// Service for ingesting data. This function block should be called on 
// every cycle to continually stream any data stored in the internal buffer.
FUNCTION_BLOCK FB_IngestService
VAR_INPUT
	hSiftClient : REFERENCE TO T_SiftClient;
	sRunId : STRING(255);
	aFlowConfigs : POINTER TO ST_FlowConfig;
END_VAR

VAR_OUTPUT
	bError : BOOL;
	nErrId : UDINT;
	nMsgsSent : UDINT; // Number of total messages sent to sift_proxy.
	nBufSize : UDINT; // The number of messages in the buffer.
	fBufferUtilization : LREAL; // The percent utilization of the internal buffer.
END_VAR

VAR
	eState : (IDLE, SEND_MESSAGE, SEND_MESSAGE_WAIT, SUCCESS, FAILURE):= IDLE;
	fbSendRingBuffer : FB_MemRingBuffer;
	aSendRingBuffer : ARRAY[0..SiftClientParameters.MAX_PACKET_SIZE - 1] OF BYTE;
	aTmpBuffer : ARRAY[0..SiftClientParameters.MAX_PACKET_SIZE - 1] OF BYTE;
	curOffset : UDINT;
	i : UDINT;
	nCount : UDINT;
END_VAR

nBufSize := fbSendRingBuffer.nCount;
fBufferUtilization := UDINT_TO_LREAL(fbSendRingBuffer.cbSize) / UDINT_TO_LREAL(SiftClientParameters.MAX_PACKET_SIZE);

CASE eState OF
	IDLE:
		bError := FALSE;
		IF nBufSize > 0 THEN
			nCount := nBufSize;
			eState := SEND_MESSAGE;
			
		END_IF
			
	SEND_MESSAGE:
		bError := FALSE;
		
		curOffset := 0;
		FOR i := 1 TO nCount DO
			fbSendRingBuffer.A_RemoveHead(pRead := ADR(aTmpBuffer[curOffset]),
										  cbRead := SiftClientParameters.MAX_PACKET_SIZE - curOffset,
										  pBuffer := ADR(aSendRingBuffer),
										  cbBuffer := SiftClientParameters.MAX_PACKET_SIZE);
			IF NOT fbSendRingBuffer.bOk THEN
				eState := FAILURE;
				nErrId := GVL_SIFT.INGEST_RING_BUFFER_REMOVE_ERROR;
				RETURN;
			END_IF
			curOffset := curOffset + fbSendRingBuffer.cbReturn;
		END_FOR
		nCount := 0;
		
		hSiftClient.fbSend(
			hSocket := hSiftClient.fbConnect.hSocket, 
			pSrc := ADR(aTmpBuffer),
			cbLen := curOffset,
			bExecute := TRUE,
		);
		
		eState := SEND_MESSAGE_WAIT;

	SEND_MESSAGE_WAIT:
		bError := FALSE;
		hSiftClient.fbSend(bExecute := FALSE);
		
		IF hSiftClient.fbSend.bBusy THEN
			RETURN;
		ELSIF hSiftClient.fbSend.bError THEN
			nErrId := hSiftClient.fbSend.nErrId;
			eState := FAILURE;
			RETURN;
		END_IF	
		
		nMsgsSent := nMsgsSent + 1;
		eState := IDLE;
		
	FAILURE:
		bError := TRUE;
END_CASE

// Writes data from a Flow to the buffer to be sent to Sift.
// This should be called for each time you want to record data
// for a given flow.
METHOD PUBLIC WriteData : BOOL
VAR_INPUT
	pFlowConfig : POINTER TO ST_FlowConfig;
	stTimestamp : _ST_Timestamp;
END_VAR

VAR_OUTPUT
	bError : BOOL;
END_VAR

VAR
	// TODO: This should be allocated on the heap (FB local var);
	aRawBuf : ARRAY[1..SiftClientParameters.MAX_PACKET_SIZE] OF BYTE;
	fbWriter : _FB_BufferWriter := (pRawBuf := ADR(aRawBuf), nSize := SIZEOF(aRawBuf));
	nMsgSize : UDINT;
END_VAR
IF pFlowConfig = 0 THEN
	WriteData := FALSE;
	RETURN;
END_IF

nMsgSize := _F_CreateDataMessage(fbWriter := fbWriter, 
							     pFlowConfig := pFlowConfig, 
								 sRunId := sRunId,
							     stTimestamp := stTimestamp);
IF nMsgSize = 0 THEN
	WriteData := FALSE;
	RETURN;
END_IF

fbSendRingBuffer.A_AddTail(pWrite := ADR(aRawBuf), 
						   cbWrite := nMsgSize + GVL_SIFT.HEADER_LENGTH, 
						   pBuffer := ADR(aSendRingBuffer), 
						   cbBuffer := SiftClientParameters.MAX_PACKET_SIZE);
						   
WriteData := fbSendRingBuffer.bOk;
END_METHOD

END_FUNCTION_BLOCK

(* stored: Version 1.1.0.1
   POU FB_IngestService: Id {3c66359b-9e66-4237-8835-89dcf998f3e0}, SpecialFunc None
   Method WriteData: Id {e66bc1ce-d5b1-4b4a-9edc-01a0ca24d04c} *)
